FUNCTION_BLOCK FB_WP
	VAR_INPUT
	Freigabe_auto			: BOOL;
	Freigabe_Deakt_auto		: BOOL;
	Betrieb_Anford_auto		: BOOL;
	Quittierung				: BOOL;
	Parameter_init			: ST_WP_Parameter;
END_VAR
VAR_OUTPUT
	{attribute 'OPC.UA.DA' := '1'}Steuerung				: ST_WP_Steuerung;	
	{attribute 'OPC.UA.DA' := '1'}Stellwert				: ST_WP_Stellwert;	
	{attribute 'OPC.UA.DA' := '1'}Zustand					: ST_WP_Zustand;
	{attribute 'OPC.UA.DA' := '1'}Parameter				: ST_WP_Parameter;	
END_VAR
VAR
	Zustandscheck			: FB_WP_Zustandscheck;
	Logik					: FB_WP_Logik;
	Ablaufsteuerung			: FB_WP_Ablaufsteuerung;
	QuitTrig				: FB_SetResetFallTrigger;
	SchreibeDaten: FB_WP_SchreibeDaten;

	OUT_Stellung				AT %Q* : BOOL;
END_VAR

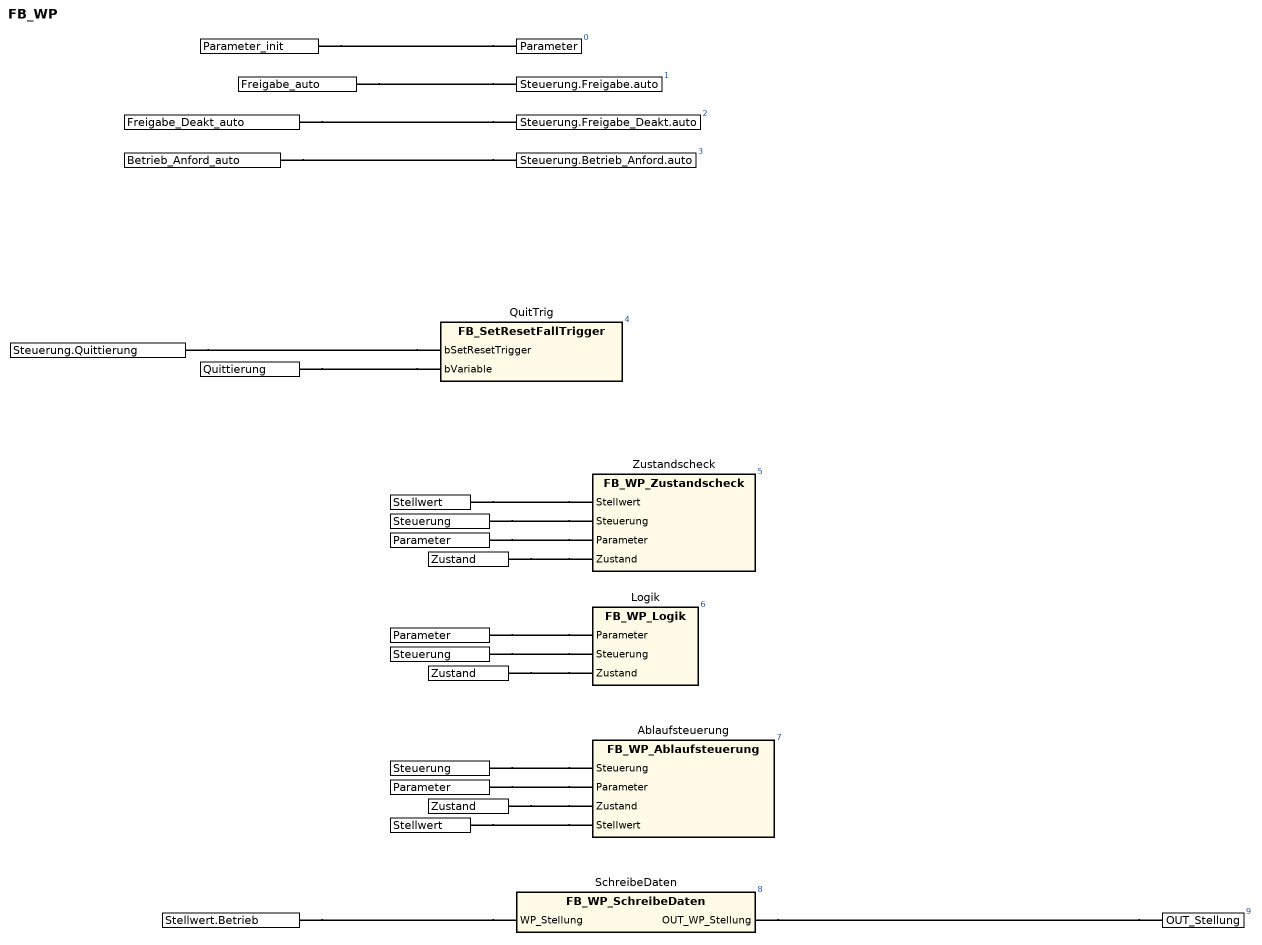
Parameter := Parameter_init;
Steuerung.Freigabe.auto := Freigabe_auto;
Steuerung.Freigabe_Deakt.auto := Freigabe_Deakt_auto;
Steuerung.Betrieb_Anford.auto := Betrieb_Anford_auto;
QuitTrig(bSetResetTrigger := Steuerung.Quittierung, bVariable := Quittierung); // FB_SetResetFallTrigger
Zustandscheck(Stellwert := Stellwert, Steuerung := Steuerung, Parameter := Parameter, Zustand := Zustand); // FB_WP_Zustandscheck
Logik(Parameter := Parameter, Steuerung := Steuerung, Zustand := Zustand); // FB_WP_Logik
Ablaufsteuerung(Steuerung := Steuerung, Parameter := Parameter, Zustand := Zustand, Stellwert := Stellwert); // FB_WP_Ablaufsteuerung
SchreibeDaten(WP_Stellung := Stellwert.Betrieb); // FB_WP_SchreibeDaten
OUT_Stellung := SchreibeDaten.OUT_WP_Stellung;

END_FUNCTION_BLOCK

(* stored: Version 1.1.0.1, ProductVersion 3.1.4024.9
   POU FB_WP: Id {7a278fbc-9761-4e22-843b-5987b4a56e4f}, SpecialFunc None *)
